// TIA Portal V21 export
FUNCTION "PRINT PV" : Void   // FC1, LAD
{ S7_Optimized_Access := 'TRUE' }
// stored: SetENOAutomatically false
   VAR_TEMP   // added for the SCL form of the ladder/FBD networks
      _w1 : Bool;
   END_VAR
BEGIN

REGION Network 1: GET DATE AND TIME
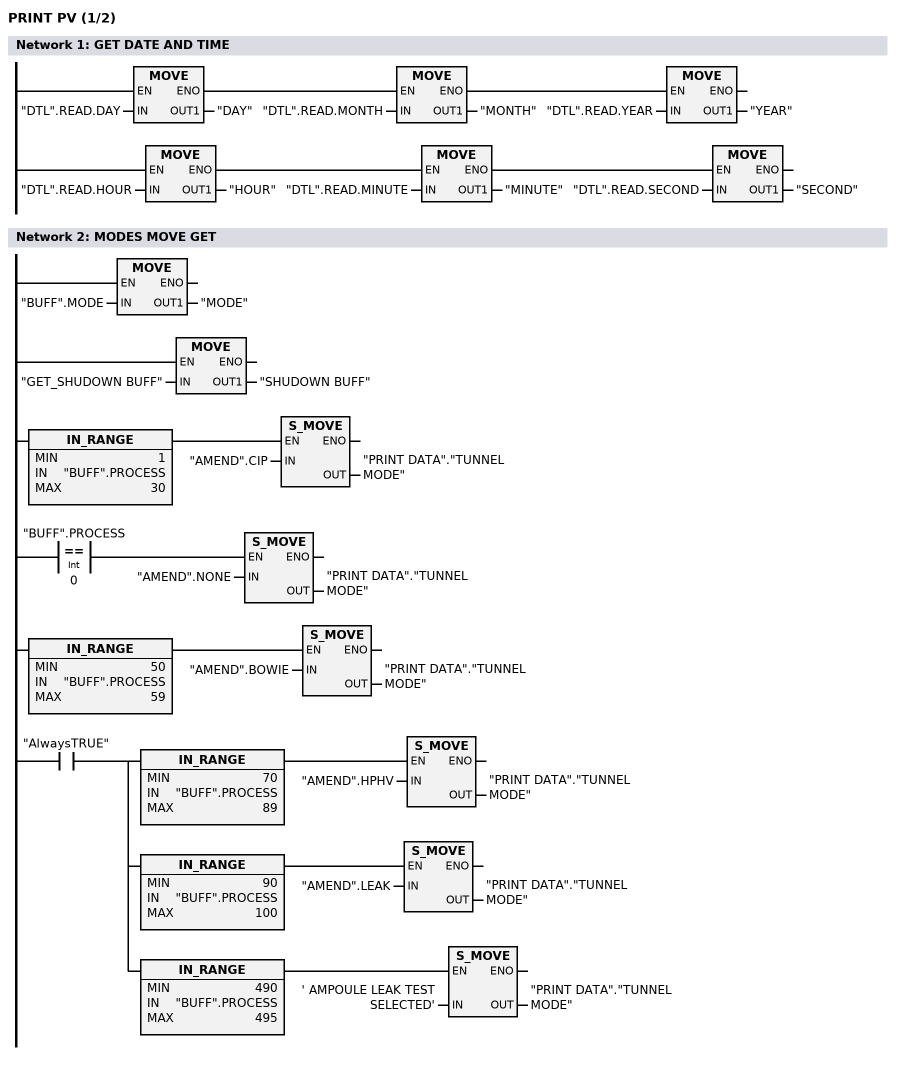
   RUNG wire#powerrail
      Move(in := "DTL".READ.DAY, out1 => "DAY")
      Move(in := "DTL".READ.MONTH, out1 => "MONTH")
      Move(in := "DTL".READ.YEAR, out1 => "YEAR")
   END_RUNG
   RUNG wire#powerrail
      Move(in := "DTL".READ.HOUR, out1 => "HOUR")
      Move(in := "DTL".READ.MINUTE, out1 => "MINUTE")
      Move(in := "DTL".READ.SECOND, out1 => "SECOND")
   END_RUNG
   // the same network as SCL:
   "DAY" := "DTL".READ.DAY;
   "MONTH" := "DTL".READ.MONTH;
   "YEAR" := "DTL".READ.YEAR;
   "HOUR" := "DTL".READ.HOUR;
   "MINUTE" := "DTL".READ.MINUTE;
   "SECOND" := "DTL".READ.SECOND;
END_REGION

REGION Network 2: MODES MOVE GET
   RUNG wire#powerrail
      Move(in := "BUFF".MODE, out1 => "MODE")
   END_RUNG
   RUNG wire#powerrail
      Move(in := "GET_SHUDOWN BUFF", out1 => "SHUDOWN BUFF")
   END_RUNG
   RUNG wire#powerrail
      { S7_Templates := "SrcType := Int" } InRange(min := 1, in := "BUFF".PROCESS, max := 30)
      S_Move(in := "AMEND".CIP, out => "PRINT DATA"."TUNNEL MODE")
   END_RUNG
   RUNG wire#powerrail
      { S7_Templates := "SrcType := Int" } EQ_Contact(in1 := "BUFF".PROCESS, in2 := 0)
      S_Move(in := "AMEND".NONE, out => "PRINT DATA"."TUNNEL MODE")
   END_RUNG
   RUNG wire#powerrail
      { S7_Templates := "SrcType := Int" } InRange(min := 50, in := "BUFF".PROCESS, max := 59)
      S_Move(in := "AMEND".BOWIE, out => "PRINT DATA"."TUNNEL MODE")
   END_RUNG
   RUNG wire#powerrail
      Contact( "AlwaysTRUE" )
      wire#w1
      { S7_Templates := "SrcType := Int" } InRange(min := 70, in := "BUFF".PROCESS, max := 89)
      S_Move(in := "AMEND".HPHV, out => "PRINT DATA"."TUNNEL MODE")
   END_RUNG
   RUNG wire#w1
      { S7_Templates := "SrcType := Int" } InRange(min := 90, in := "BUFF".PROCESS, max := 100)
      S_Move(in := "AMEND".LEAK, out => "PRINT DATA"."TUNNEL MODE")
   END_RUNG
   RUNG wire#w1
      { S7_Templates := "SrcType := Int" } InRange(min := 490, in := "BUFF".PROCESS, max := 495)
      S_Move(in := ' AMPOULE LEAK TEST SELECTED', out => "PRINT DATA"."TUNNEL MODE")
   END_RUNG
   // the same network as SCL:
   "MODE" := "BUFF".MODE;
   "SHUDOWN BUFF" := "GET_SHUDOWN BUFF";
   IF (1 <= "BUFF".PROCESS) AND ("BUFF".PROCESS <= 30) THEN
       "PRINT DATA"."TUNNEL MODE" := "AMEND".CIP;
   END_IF;
   IF "BUFF".PROCESS = 0 THEN "PRINT DATA"."TUNNEL MODE" := "AMEND".NONE; END_IF;
   IF (50 <= "BUFF".PROCESS) AND ("BUFF".PROCESS <= 59) THEN
       "PRINT DATA"."TUNNEL MODE" := "AMEND".BOWIE;
   END_IF;
   IF "AlwaysTRUE" AND (70 <= "BUFF".PROCESS) AND ("BUFF".PROCESS <= 89) THEN
       "PRINT DATA"."TUNNEL MODE" := "AMEND".HPHV;
   END_IF;
   IF "AlwaysTRUE" AND (90 <= "BUFF".PROCESS) AND ("BUFF".PROCESS <= 100) THEN
       "PRINT DATA"."TUNNEL MODE" := "AMEND".LEAK;
   END_IF;
   IF "AlwaysTRUE" AND (490 <= "BUFF".PROCESS) AND ("BUFF".PROCESS <= 495) THEN
       "PRINT DATA"."TUNNEL MODE" := ' AMPOULE LEAK TEST SELECTED';
   END_IF;
END_REGION

REGION Network 3
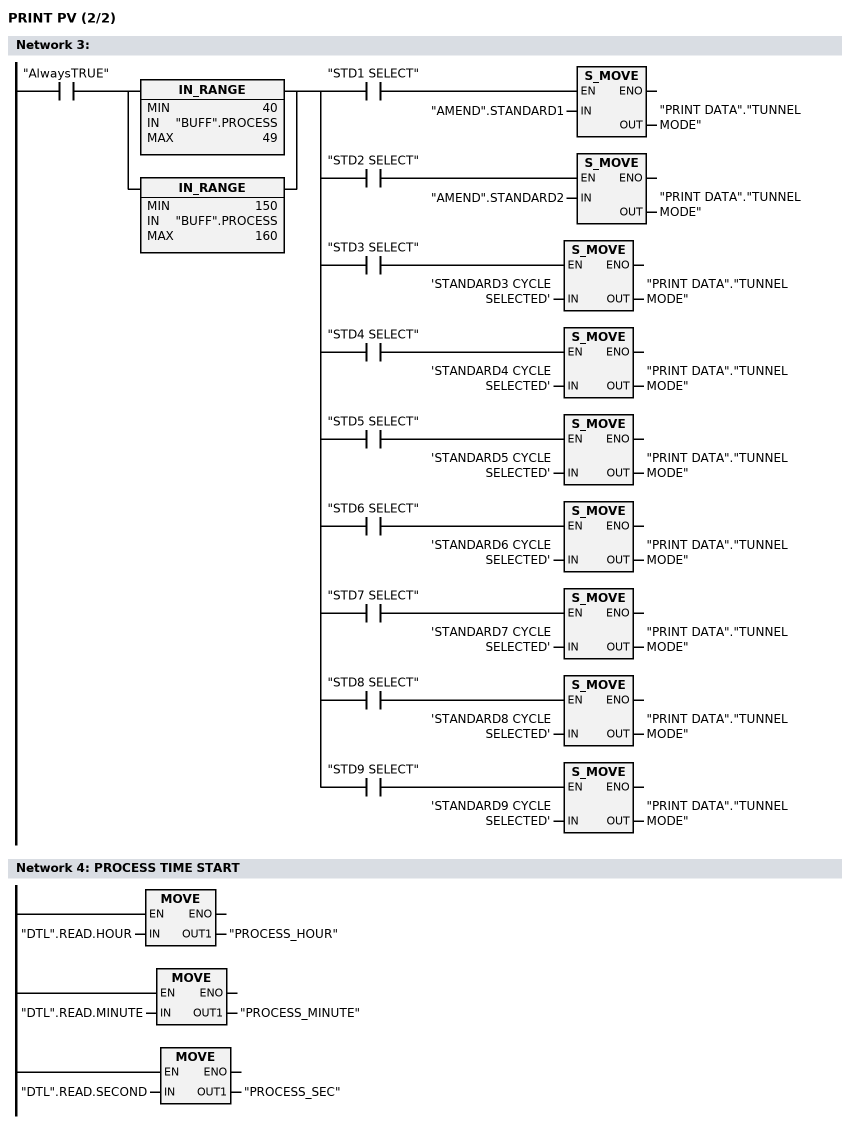
   RUNG wire#powerrail
      Contact( "AlwaysTRUE" )
      wire#w1
      { S7_Templates := "SrcType := Int" } InRange(min := 40, in := "BUFF".PROCESS, max := 49)
      wire#w2
      Contact( "STD1 SELECT" )
      S_Move(in := "AMEND".STANDARD1, out => "PRINT DATA"."TUNNEL MODE")
   END_RUNG
   RUNG wire#w1
      { S7_Templates := "SrcType := Int" } InRange(min := 150, in := "BUFF".PROCESS, max := 160)
   END_RUNG wire#w2
   RUNG wire#w2
      Contact( "STD2 SELECT" )
      S_Move(in := "AMEND".STANDARD2, out => "PRINT DATA"."TUNNEL MODE")
   END_RUNG
   RUNG wire#w2
      Contact( "STD3 SELECT" )
      S_Move(in := 'STANDARD3 CYCLE SELECTED', out => "PRINT DATA"."TUNNEL MODE")
   END_RUNG
   RUNG wire#w2
      Contact( "STD4 SELECT" )
      S_Move(in := 'STANDARD4 CYCLE SELECTED', out => "PRINT DATA"."TUNNEL MODE")
   END_RUNG
   RUNG wire#w2
      Contact( "STD5 SELECT" )
      S_Move(in := 'STANDARD5 CYCLE SELECTED', out => "PRINT DATA"."TUNNEL MODE")
   END_RUNG
   RUNG wire#w2
      Contact( "STD6 SELECT" )
      S_Move(in := 'STANDARD6 CYCLE SELECTED', out => "PRINT DATA"."TUNNEL MODE")
   END_RUNG
   RUNG wire#w2
      Contact( "STD7 SELECT" )
      S_Move(in := 'STANDARD7 CYCLE SELECTED', out => "PRINT DATA"."TUNNEL MODE")
   END_RUNG
   RUNG wire#w2
      Contact( "STD8 SELECT" )
      S_Move(in := 'STANDARD8 CYCLE SELECTED', out => "PRINT DATA"."TUNNEL MODE")
   END_RUNG
   RUNG wire#w2
      Contact( "STD9 SELECT" )
      S_Move(in := 'STANDARD9 CYCLE SELECTED', out => "PRINT DATA"."TUNNEL MODE")
   END_RUNG
   // the same network as SCL:
   #_w1 := "AlwaysTRUE" AND (((40 <= "BUFF".PROCESS) AND ("BUFF".PROCESS <= 49)) OR ((150 <= "BUFF".PROCESS) AND ("BUFF".PROCESS <= 160)));
   IF #_w1 AND "STD1 SELECT" THEN "PRINT DATA"."TUNNEL MODE" := "AMEND".STANDARD1; END_IF;
   IF #_w1 AND "STD2 SELECT" THEN "PRINT DATA"."TUNNEL MODE" := "AMEND".STANDARD2; END_IF;
   IF #_w1 AND "STD3 SELECT" THEN "PRINT DATA"."TUNNEL MODE" := 'STANDARD3 CYCLE SELECTED'; END_IF;
   IF #_w1 AND "STD4 SELECT" THEN "PRINT DATA"."TUNNEL MODE" := 'STANDARD4 CYCLE SELECTED'; END_IF;
   IF #_w1 AND "STD5 SELECT" THEN "PRINT DATA"."TUNNEL MODE" := 'STANDARD5 CYCLE SELECTED'; END_IF;
   IF #_w1 AND "STD6 SELECT" THEN "PRINT DATA"."TUNNEL MODE" := 'STANDARD6 CYCLE SELECTED'; END_IF;
   IF #_w1 AND "STD7 SELECT" THEN "PRINT DATA"."TUNNEL MODE" := 'STANDARD7 CYCLE SELECTED'; END_IF;
   IF #_w1 AND "STD8 SELECT" THEN "PRINT DATA"."TUNNEL MODE" := 'STANDARD8 CYCLE SELECTED'; END_IF;
   IF #_w1 AND "STD9 SELECT" THEN "PRINT DATA"."TUNNEL MODE" := 'STANDARD9 CYCLE SELECTED'; END_IF;
END_REGION

REGION Network 4: PROCESS TIME START
   RUNG wire#powerrail
      Move(in := "DTL".READ.HOUR, out1 => "PROCESS_HOUR")
   END_RUNG
   RUNG wire#powerrail
      Move(in := "DTL".READ.MINUTE, out1 => "PROCESS_MINUTE")
   END_RUNG
   RUNG wire#powerrail
      Move(in := "DTL".READ.SECOND, out1 => "PROCESS_SEC")
   END_RUNG
   // the same network as SCL:
   "PROCESS_HOUR" := "DTL".READ.HOUR;
   "PROCESS_MINUTE" := "DTL".READ.MINUTE;
   "PROCESS_SEC" := "DTL".READ.SECOND;
END_REGION
END_FUNCTION
